PROGRAM MAIN
VAR
	fbSR : SR;
END_VAR

fbSR(SET1:= GVL.bDigital_Inputs[1], RESET:= GVL.bDigital_Inputs[2]);

GVL.bDigital_Outputs[1] := fbSR.Q1;
GVL.bDigital_Outputs[2] := fbSR.Q1;
GVL.bDigital_Outputs[3] := fbSR.Q1;
GVL.bDigital_Outputs[4] := fbSR.Q1;
GVL.bDigital_Outputs[5] := fbSR.Q1;
GVL.bDigital_Outputs[6] := fbSR.Q1;

END_PROGRAM

(* stored: Version 1.1.0.1, ProductVersion 3.1.4024.12
   POU MAIN: Id {ba39c786-a621-4770-bc5d-4d67f5182d72}, SpecialFunc None *)
